PROGRAM Plc_Prog
VAR
	Motor1 : Motor;
	Motor2 : Motor;
	Motor3 : Motor;
	
	Motor1Variables : MotorVariables;
	Motor2Variables : MotorVariables;
	Motor3Variables : MotorVariables;
END_VAR

Motor1(Start:=Motor1Variables.Start, Stop:=Motor1Variables.Stop, Overload:=Motor1Variables.Oveload, Coil=>Motor1Variables.Coil);
Motor2(Start:=Motor2Variables.Start, Stop:=Motor2Variables.Stop, Overload:=Motor2Variables.Oveload, Coil=>Motor2Variables.Coil);
Motor3(Start:=Motor3Variables.Start, Stop:=Motor3Variables.Stop, Overload:=Motor3Variables.Oveload, Coil=>Motor3Variables.Coil);

END_PROGRAM

(* stored: Version 1.1.0.1, ProductVersion 3.1.4024.9
   POU Plc_Prog: Id {71382d43-d085-4a03-b6d4-ff32041d5c6a}, SpecialFunc None *)
